// TIA Portal V20 export
DATA_BLOCK "DiagnosticsSignalsInterface"   // DB138
// stored: MemoryReserve 100
   VAR
      SignalsInterface { S7_SetPoint := 'True'} : "LER_SignalsInterface";
   END_VAR
BEGIN
   SignalsInterface.HMI_Select_Mode := FALSE;
   SignalsInterface.ButtonValue[0].ButtonLeft[0..15] := FALSE;
   SignalsInterface.ButtonValue[1].ButtonLeft[0..15] := FALSE;
   SignalsInterface.ButtonValue[2].ButtonLeft[0..15] := FALSE;
   SignalsInterface.ButtonValue[3].ButtonLeft[0..15] := FALSE;
   SignalsInterface.ButtonValue[4].ButtonLeft[0..15] := FALSE;
   SignalsInterface.ButtonValue[5].ButtonLeft[0..15] := FALSE;
   SignalsInterface.ButtonValue[6].ButtonLeft[0..15] := FALSE;
   SignalsInterface.ButtonValue[7].ButtonLeft[0..15] := FALSE;
   SignalsInterface.ButtonValue[8].ButtonLeft[0..15] := FALSE;
   SignalsInterface.ButtonValue[9].ButtonLeft[0..15] := FALSE;
   SignalsInterface.ButtonValue[10].ButtonLeft[0..15] := FALSE;
   SignalsInterface.ButtonValue[11].ButtonLeft[0..15] := FALSE;
   SignalsInterface.ButtonValue[12].ButtonLeft[0..15] := FALSE;
   SignalsInterface.ButtonValue[13].ButtonLeft[0..15] := FALSE;
   SignalsInterface.ButtonValue[14].ButtonLeft[0..15] := FALSE;
   SignalsInterface.ButtonValue[15].ButtonLeft[0..15] := FALSE;
   SignalsInterface.ButtonValue[16].ButtonLeft[0..15] := FALSE;
   SignalsInterface.ButtonValue[0].ButtonRight[0..15] := FALSE;
   SignalsInterface.ButtonValue[1].ButtonRight[0..15] := FALSE;
   SignalsInterface.ButtonValue[2].ButtonRight[0..15] := FALSE;
   SignalsInterface.ButtonValue[3].ButtonRight[0..15] := FALSE;
   SignalsInterface.ButtonValue[4].ButtonRight[0..15] := FALSE;
   SignalsInterface.ButtonValue[5].ButtonRight[0..15] := FALSE;
   SignalsInterface.ButtonValue[6].ButtonRight[0..15] := FALSE;
   SignalsInterface.ButtonValue[7].ButtonRight[0..15] := FALSE;
   SignalsInterface.ButtonValue[8].ButtonRight[0..15] := FALSE;
   SignalsInterface.ButtonValue[9].ButtonRight[0..15] := FALSE;
   SignalsInterface.ButtonValue[10].ButtonRight[0..15] := FALSE;
   SignalsInterface.ButtonValue[11].ButtonRight[0..15] := FALSE;
   SignalsInterface.ButtonValue[12].ButtonRight[0..15] := FALSE;
   SignalsInterface.ButtonValue[13].ButtonRight[0..15] := FALSE;
   SignalsInterface.ButtonValue[14].ButtonRight[0..15] := FALSE;
   SignalsInterface.ButtonValue[15].ButtonRight[0..15] := FALSE;
   SignalsInterface.ButtonValue[16].ButtonRight[0..15] := FALSE;
END_DATA_BLOCK
